{attribute addProperty BoxType "EJ2914-0000-0017"}
{attribute addProperty Id "Module_1_FSOEModule_1_FSOE_D19648F396120Module_2_FSOUTModule_2_FSOUT_B889B7D03240Module_3_DEVICEIOModule_3_DEVICEIO_FB2B67D71620Module_4_FSLOGICModule_4_FSLOGIC_3E6251391620WcStateAT %I*WcState_C1B70B0F3240InfoDataAT %I*InfoData_BC63D37F80100"}
{attribute addProperty CRC "2197355110"}
{attribute addProperty SizeInBites "272"}
{attribute addProperty SizeInBytes "34"}
TYPE EJ2914_26D491F1 :
STRUCT
	{attribute addProperty Name "Module_1_FSOE"}
	Module_1_FSOE : Module_1_FSOE_D19648F3;
	{attribute addProperty Name "Module_2_FSOUT"}
	Module_2_FSOUT : Module_2_FSOUT_B889B7D0;
	{attribute addProperty Name "Module_3_DEVICEIO"}
	Module_3_DEVICEIO : Module_3_DEVICEIO_FB2B67D7;
	{attribute addProperty Name "Module_4_FSLOGIC"}
	Module_4_FSLOGIC : Module_4_FSLOGIC_3E625139;
	{attribute addProperty Name "WcState"}
	WcState : WcState_C1B70B0F;
	{attribute addProperty Name "InfoData"}
	InfoData : InfoData_BC63D37F;
END_STRUCT
END_TYPE

(* stored: Version 1.2.0.0, ProductVersion 3.1.4024.9
   DUT EJ2914_26D491F1: Id {f71a15a6-6976-473d-a800-99ed699707a6} *)
